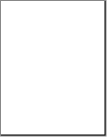
VISUALIZATION VISU_EtherCatFillerDevice  // 107x137
    Rectangle (0,0 105x135)
END_VISUALIZATION

(* stored: Version 1.1.0.1, ProductVersion 3.1.0.36
   Visu VISU_EtherCatFillerDevice: Id {b3d9ca70-1047-48a7-975f-7478cb9858e7} *)
